{attribute addProperty BoxType "EJ7334-0008-0016"}
{attribute addProperty Id "ControlAT %Q*Control_96E4A9881621VelocityAT %Q*INT16233"}
{attribute addProperty CRC "527943874"}
{attribute addProperty SizeInBites "32"}
{attribute addProperty SizeInBytes "4"}
TYPE DCM_Outputs_Channel_1F77C8C2 :
STRUCT
	{attribute addProperty Name "Control"}
	Control AT %Q* : Control_96E4A988;
	{attribute addProperty Name "Velocity"}
	Velocity AT %Q* : INT;
END_STRUCT
END_TYPE

(* stored: Version 1.2.0.0, ProductVersion 3.1.4024.9
   DUT DCM_Outputs_Channel_1F77C8C2: Id {7699cbb7-f728-48f4-a38c-b54abd2d59a4} *)
